PROGRAM MAIN
VAR
	
END_VAR


P_Safety();						// Check doors, safety switches etc. before going through with main program

IF GENERAL.ReadyForAction AND SAFETY.Safety_OK THEN 	// If both signals indicating readyness are given, go through with main tasks.
		P_BACKGROUND();					// Background routines. Blinks etc
		P_WritePersistentData();		// Writes persistent variables to memory every 10 seconds
		OVERVIEW_FBD();					// FBD View of all FB's. Useful visualization of whats happening
			// P_Environment_Control 		-> Is a separate slow task, not to be called from MAIN
END_IF

END_PROGRAM

(* stored: Version 1.1.0.1, ProductVersion 3.1.4024.10
   POU MAIN: Id {9ad04803-898f-4588-9872-113a1d3cdead}, SpecialFunc None *)
